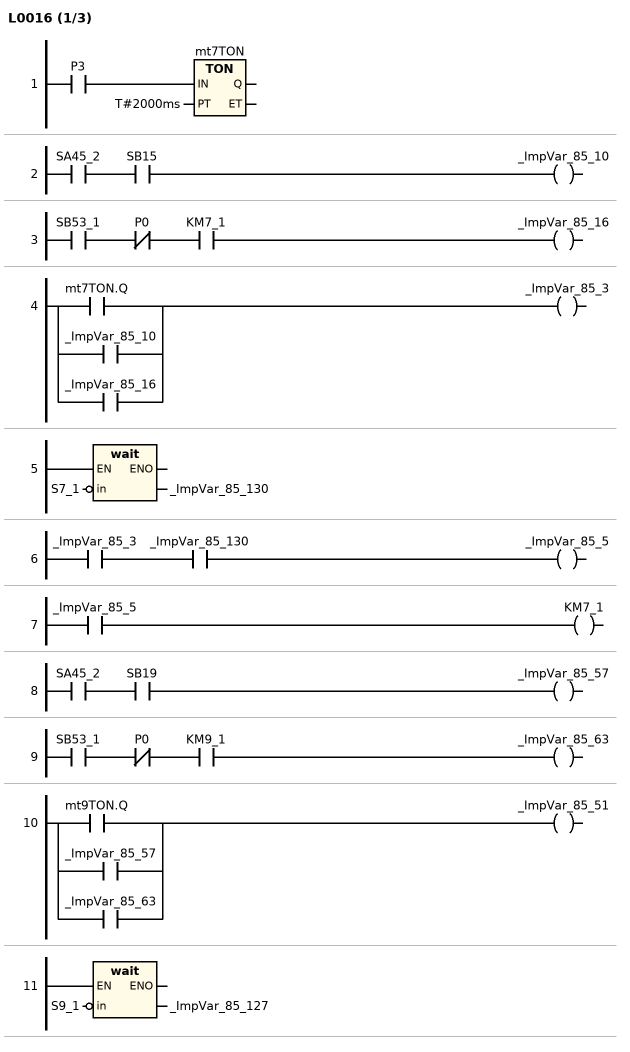
[picture p24: L0016 (LD)]
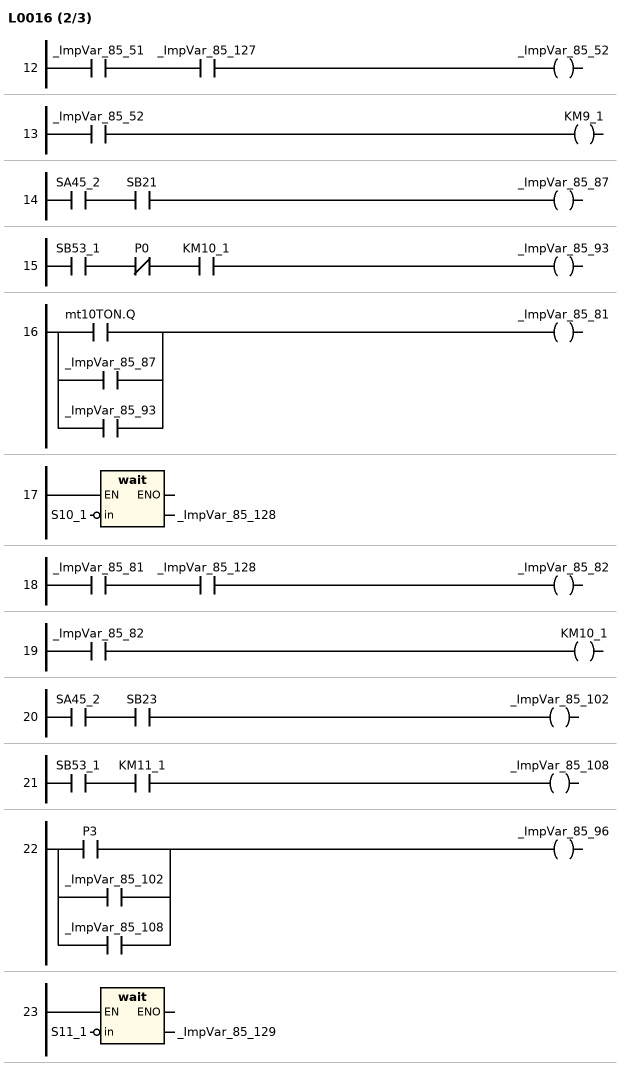
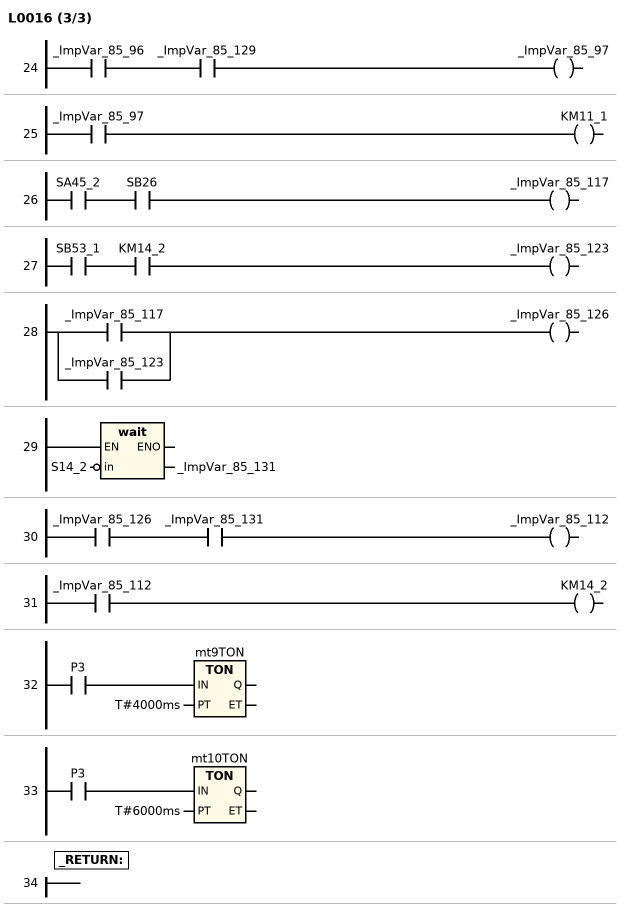
_LD_ (* Ladder Diagram *)
NETWORK 1
	[P3] - mt7TON:TON(IN: *, PT: T#2000ms)
NETWORK 2
	[SA45_2] - [SB15] --- (_ImpVar_85_10)
NETWORK 3
	[SB53_1] - [/P0] - [KM7_1] --- (_ImpVar_85_16)
NETWORK 4
	{ [mt7TON.Q] | [_ImpVar_85_10] | [_ImpVar_85_16] } --- (_ImpVar_85_3)
NETWORK 5
	*
		EN --- wait(in: NOT S7_1) => _ImpVar_85_130
NETWORK 6
	[_ImpVar_85_3] - [_ImpVar_85_130] --- (_ImpVar_85_5)
NETWORK 7
	[_ImpVar_85_5] --- (KM7_1)
NETWORK 8
	[SA45_2] - [SB19] --- (_ImpVar_85_57)
NETWORK 9
	[SB53_1] - [/P0] - [KM9_1] --- (_ImpVar_85_63)
NETWORK 10
	{ [mt9TON.Q] | [_ImpVar_85_57] | [_ImpVar_85_63] } --- (_ImpVar_85_51)
NETWORK 11
	*
		EN --- wait(in: NOT S9_1) => _ImpVar_85_127
NETWORK 12
	[_ImpVar_85_51] - [_ImpVar_85_127] --- (_ImpVar_85_52)
NETWORK 13
	[_ImpVar_85_52] --- (KM9_1)
NETWORK 14
	[SA45_2] - [SB21] --- (_ImpVar_85_87)
NETWORK 15
	[SB53_1] - [/P0] - [KM10_1] --- (_ImpVar_85_93)
NETWORK 16
	{ [mt10TON.Q] | [_ImpVar_85_87] | [_ImpVar_85_93] } --- (_ImpVar_85_81)
NETWORK 17
	*
		EN --- wait(in: NOT S10_1) => _ImpVar_85_128
NETWORK 18
	[_ImpVar_85_81] - [_ImpVar_85_128] --- (_ImpVar_85_82)
NETWORK 19
	[_ImpVar_85_82] --- (KM10_1)
NETWORK 20
	[SA45_2] - [SB23] --- (_ImpVar_85_102)
NETWORK 21
	[SB53_1] - [KM11_1] --- (_ImpVar_85_108)
NETWORK 22
	{ [P3] | [_ImpVar_85_102] | [_ImpVar_85_108] } --- (_ImpVar_85_96)
NETWORK 23
	*
		EN --- wait(in: NOT S11_1) => _ImpVar_85_129
NETWORK 24
	[_ImpVar_85_96] - [_ImpVar_85_129] --- (_ImpVar_85_97)
NETWORK 25
	[_ImpVar_85_97] --- (KM11_1)
NETWORK 26
	[SA45_2] - [SB26] --- (_ImpVar_85_117)
NETWORK 27
	[SB53_1] - [KM14_2] --- (_ImpVar_85_123)
NETWORK 28
	{ [_ImpVar_85_117] | [_ImpVar_85_123] } --- (_ImpVar_85_126)
NETWORK 29
	*
		EN --- wait(in: NOT S14_2) => _ImpVar_85_131
NETWORK 30
	[_ImpVar_85_126] - [_ImpVar_85_131] --- (_ImpVar_85_112)
NETWORK 31
	[_ImpVar_85_112] --- (KM14_2)
NETWORK 32
	[P3] - mt9TON:TON(IN: *, PT: T#4000ms)
NETWORK 33
	[P3] - mt10TON:TON(IN: *, PT: T#6000ms)
NETWORK 34 _RETURN::
	*
_END_LD_
(* the same logic as Structured Text *)
(* Network 1 *)
mt7TON(IN := P3, PT := T#2000ms);
(* Network 2 *)
_ImpVar_85_10 := SA45_2 AND SB15;
(* Network 3 *)
_ImpVar_85_16 := SB53_1 AND NOT P0 AND KM7_1;
(* Network 4 *)
_ImpVar_85_3 := mt7TON.Q OR _ImpVar_85_10 OR _ImpVar_85_16;
(* Network 5 *)
_ImpVar_85_130 := wait(in := NOT S7_1);
(* Network 6 *)
_ImpVar_85_5 := _ImpVar_85_3 AND _ImpVar_85_130;
(* Network 7 *)
KM7_1 := _ImpVar_85_5;
(* Network 8 *)
_ImpVar_85_57 := SA45_2 AND SB19;
(* Network 9 *)
_ImpVar_85_63 := SB53_1 AND NOT P0 AND KM9_1;
(* Network 10 *)
_ImpVar_85_51 := mt9TON.Q OR _ImpVar_85_57 OR _ImpVar_85_63;
(* Network 11 *)
_ImpVar_85_127 := wait(in := NOT S9_1);
(* Network 12 *)
_ImpVar_85_52 := _ImpVar_85_51 AND _ImpVar_85_127;
(* Network 13 *)
KM9_1 := _ImpVar_85_52;
(* Network 14 *)
_ImpVar_85_87 := SA45_2 AND SB21;
(* Network 15 *)
_ImpVar_85_93 := SB53_1 AND NOT P0 AND KM10_1;
(* Network 16 *)
_ImpVar_85_81 := mt10TON.Q OR _ImpVar_85_87 OR _ImpVar_85_93;
(* Network 17 *)
_ImpVar_85_128 := wait(in := NOT S10_1);
(* Network 18 *)
_ImpVar_85_82 := _ImpVar_85_81 AND _ImpVar_85_128;
(* Network 19 *)
KM10_1 := _ImpVar_85_82;
(* Network 20 *)
_ImpVar_85_102 := SA45_2 AND SB23;
(* Network 21 *)
_ImpVar_85_108 := SB53_1 AND KM11_1;
(* Network 22 *)
_ImpVar_85_96 := P3 OR _ImpVar_85_102 OR _ImpVar_85_108;
(* Network 23 *)
_ImpVar_85_129 := wait(in := NOT S11_1);
(* Network 24 *)
_ImpVar_85_97 := _ImpVar_85_96 AND _ImpVar_85_129;
(* Network 25 *)
KM11_1 := _ImpVar_85_97;
(* Network 26 *)
_ImpVar_85_117 := SA45_2 AND SB26;
(* Network 27 *)
_ImpVar_85_123 := SB53_1 AND KM14_2;
(* Network 28 *)
_ImpVar_85_126 := _ImpVar_85_117 OR _ImpVar_85_123;
(* Network 29 *)
_ImpVar_85_131 := wait(in := NOT S14_2);
(* Network 30 *)
_ImpVar_85_112 := _ImpVar_85_126 AND _ImpVar_85_131;
(* Network 31 *)
KM14_2 := _ImpVar_85_112;
(* Network 32 *)
mt9TON(IN := P3, PT := T#4000ms);
(* Network 33 *)
mt10TON(IN := P3, PT := T#6000ms);
(* Network 34 *)
(* label: _RETURN: *)
END_PROGRAM

(* POU gatesAlarm, LD *)
PROGRAM gatesAlarm
VAR
	al1: alarm;
	al18_2: alarm;
	al18_1: alarm;
	al4_1: alarm;
	al4_2: alarm;
	al5_1: alarm;
	al5_2: alarm;
	al6_1: alarm;
	al6_2: alarm;
	al7_2: alarm;
	al7_1: alarm;
	al8_1: alarm;
	al8_2: alarm;
	al9_1: alarm;
	al9_2: alarm;
	al10_1: alarm;
	al10_2: alarm;
	a11_1: alarm;
	al11_2: alarm;
	al14_1: alarm;
	al14_2: alarm;
	vaqt : WORD := 70;
END_VAR
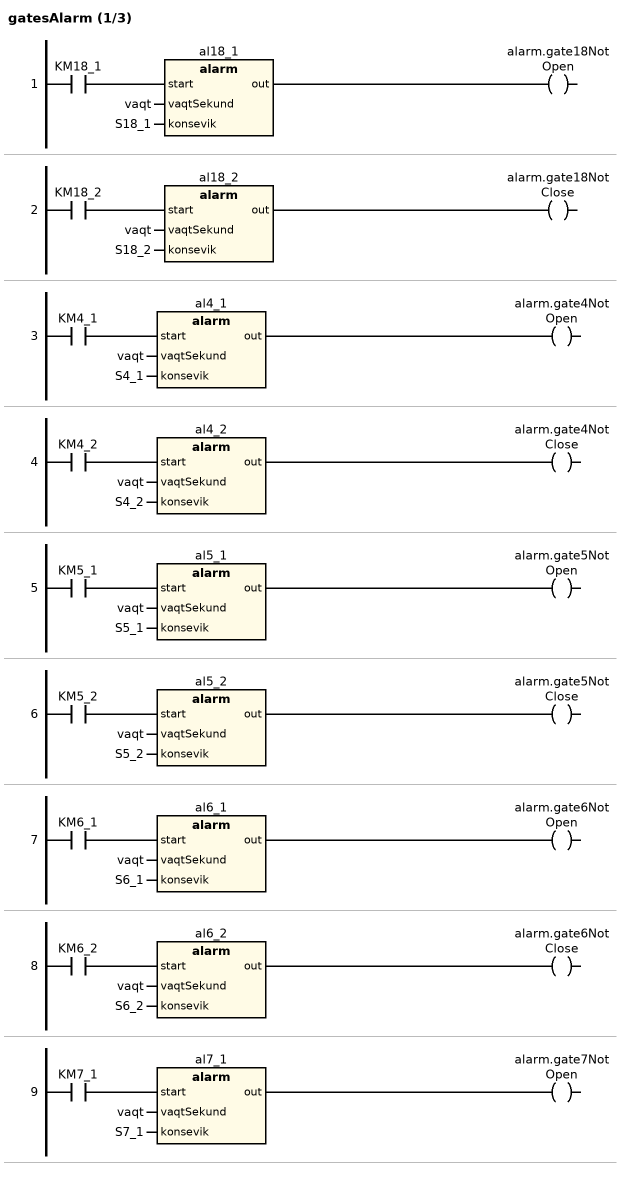
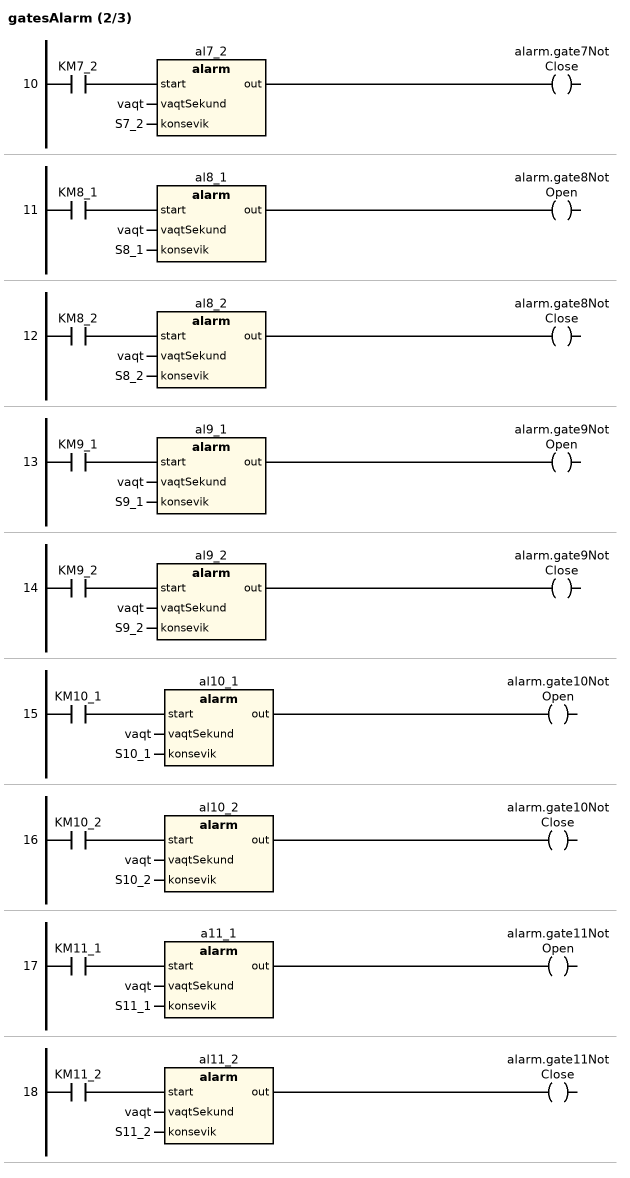
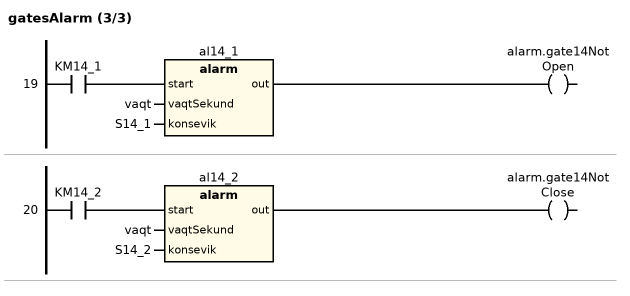
_LD_ (* Ladder Diagram *)
NETWORK 1
	[KM18_1] - al18_1:alarm(start: *, vaqtSekund: vaqt, konsevik: S18_1) --- (alarm.gate18NotOpen)
NETWORK 2
	[KM18_2] - al18_2:alarm(start: *, vaqtSekund: vaqt, konsevik: S18_2) --- (alarm.gate18NotClose)
NETWORK 3
	[KM4_1] - al4_1:alarm(start: *, vaqtSekund: vaqt, konsevik: S4_1) --- (alarm.gate4NotOpen)
NETWORK 4
	[KM4_2] - al4_2:alarm(start: *, vaqtSekund: vaqt, konsevik: S4_2) --- (alarm.gate4NotClose)
NETWORK 5
	[KM5_1] - al5_1:alarm(start: *, vaqtSekund: vaqt, konsevik: S5_1) --- (alarm.gate5NotOpen)
NETWORK 6
	[KM5_2] - al5_2:alarm(start: *, vaqtSekund: vaqt, konsevik: S5_2) --- (alarm.gate5NotClose)
NETWORK 7
	[KM6_1] - al6_1:alarm(start: *, vaqtSekund: vaqt, konsevik: S6_1) --- (alarm.gate6NotOpen)
NETWORK 8
	[KM6_2] - al6_2:alarm(start: *, vaqtSekund: vaqt, konsevik: S6_2) --- (alarm.gate6NotClose)
NETWORK 9
	[KM7_1] - al7_1:alarm(start: *, vaqtSekund: vaqt, konsevik: S7_1) --- (alarm.gate7NotOpen)
NETWORK 10
	[KM7_2] - al7_2:alarm(start: *, vaqtSekund: vaqt, konsevik: S7_2) --- (alarm.gate7NotClose)
NETWORK 11
	[KM8_1] - al8_1:alarm(start: *, vaqtSekund: vaqt, konsevik: S8_1) --- (alarm.gate8NotOpen)
NETWORK 12
	[KM8_2] - al8_2:alarm(start: *, vaqtSekund: vaqt, konsevik: S8_2) --- (alarm.gate8NotClose)
NETWORK 13
	[KM9_1] - al9_1:alarm(start: *, vaqtSekund: vaqt, konsevik: S9_1) --- (alarm.gate9NotOpen)
NETWORK 14
	[KM9_2] - al9_2:alarm(start: *, vaqtSekund: vaqt, konsevik: S9_2) --- (alarm.gate9NotClose)
NETWORK 15
	[KM10_1] - al10_1:alarm(start: *, vaqtSekund: vaqt, konsevik: S10_1) --- (alarm.gate10NotOpen)
NETWORK 16
	[KM10_2] - al10_2:alarm(start: *, vaqtSekund: vaqt, konsevik: S10_2) --- (alarm.gate10NotClose)
NETWORK 17
	[KM11_1] - a11_1:alarm(start: *, vaqtSekund: vaqt, konsevik: S11_1) --- (alarm.gate11NotOpen)
NETWORK 18
	[KM11_2] - al11_2:alarm(start: *, vaqtSekund: vaqt, konsevik: S11_2) --- (alarm.gate11NotClose)
NETWORK 19
	[KM14_1] - al14_1:alarm(start: *, vaqtSekund: vaqt, konsevik: S14_1) --- (alarm.gate14NotOpen)
NETWORK 20
	[KM14_2] - al14_2:alarm(start: *, vaqtSekund: vaqt, konsevik: S14_2) --- (alarm.gate14NotClose)
_END_LD_
(* the same logic as Structured Text *)
(* Network 1 *)
al18_1(start := KM18_1, vaqtSekund := vaqt, konsevik := S18_1);
alarm.gate18NotOpen := al18_1.out;
(* Network 2 *)
al18_2(start := KM18_2, vaqtSekund := vaqt, konsevik := S18_2);
alarm.gate18NotClose := al18_2.out;
(* Network 3 *)
al4_1(start := KM4_1, vaqtSekund := vaqt, konsevik := S4_1);
alarm.gate4NotOpen := al4_1.out;
(* Network 4 *)
al4_2(start := KM4_2, vaqtSekund := vaqt, konsevik := S4_2);
alarm.gate4NotClose := al4_2.out;
(* Network 5 *)
al5_1(start := KM5_1, vaqtSekund := vaqt, konsevik := S5_1);
alarm.gate5NotOpen := al5_1.out;
(* Network 6 *)
al5_2(start := KM5_2, vaqtSekund := vaqt, konsevik := S5_2);
alarm.gate5NotClose := al5_2.out;
(* Network 7 *)
al6_1(start := KM6_1, vaqtSekund := vaqt, konsevik := S6_1);
alarm.gate6NotOpen := al6_1.out;
(* Network 8 *)
al6_2(start := KM6_2, vaqtSekund := vaqt, konsevik := S6_2);
alarm.gate6NotClose := al6_2.out;
(* Network 9 *)
al7_1(start := KM7_1, vaqtSekund := vaqt, konsevik := S7_1);
alarm.gate7NotOpen := al7_1.out;
(* Network 10 *)
al7_2(start := KM7_2, vaqtSekund := vaqt, konsevik := S7_2);
alarm.gate7NotClose := al7_2.out;
(* Network 11 *)
al8_1(start := KM8_1, vaqtSekund := vaqt, konsevik := S8_1);
alarm.gate8NotOpen := al8_1.out;
(* Network 12 *)
al8_2(start := KM8_2, vaqtSekund := vaqt, konsevik := S8_2);
alarm.gate8NotClose := al8_2.out;
(* Network 13 *)
al9_1(start := KM9_1, vaqtSekund := vaqt, konsevik := S9_1);
alarm.gate9NotOpen := al9_1.out;
(* Network 14 *)
al9_2(start := KM9_2, vaqtSekund := vaqt, konsevik := S9_2);
alarm.gate9NotClose := al9_2.out;
(* Network 15 *)
al10_1(start := KM10_1, vaqtSekund := vaqt, konsevik := S10_1);
alarm.gate10NotOpen := al10_1.out;
(* Network 16 *)
al10_2(start := KM10_2, vaqtSekund := vaqt, konsevik := S10_2);
alarm.gate10NotClose := al10_2.out;
(* Network 17 *)
a11_1(start := KM11_1, vaqtSekund := vaqt, konsevik := S11_1);
alarm.gate11NotOpen := a11_1.out;
(* Network 18 *)
al11_2(start := KM11_2, vaqtSekund := vaqt, konsevik := S11_2);
alarm.gate11NotClose := al11_2.out;
(* Network 19 *)
al14_1(start := KM14_1, vaqtSekund := vaqt, konsevik := S14_1);
alarm.gate14NotOpen := al14_1.out;
(* Network 20 *)
al14_2(start := KM14_2, vaqtSekund := vaqt, konsevik := S14_2);
alarm.gate14NotClose := al14_2.out;
END_PROGRAM

(* POU start_or_stop, LD *)
PROGRAM start_or_stop
VAR
	_controlFazaDI46: BOOL;
	kompressorOFF: TP;
	kompressorON: TP;
	_currentHighJD5DI00000: BOOL;
	P300000: BOOL;
	P00000: BOOL;

	alarmLedDO_MB555: BOOL;
	_kompOffDO_55555555: BOOL;
	_kompOnDO_555555: BOOL;
	trig: R_TRIG;

END_VAR
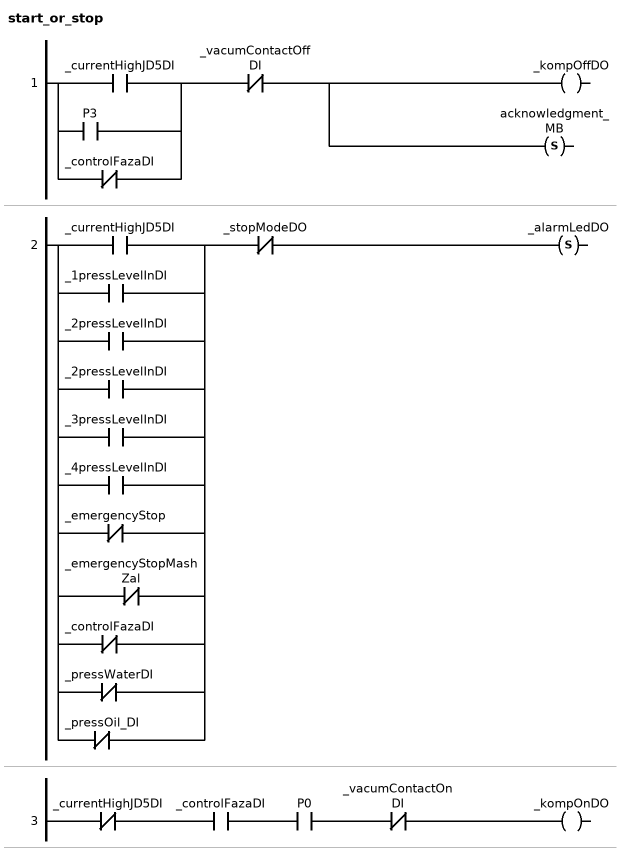
_LD_ (* Ladder Diagram *)
NETWORK 1
	{ [_currentHighJD5DI] | [P3] | [/_controlFazaDI] } - [/_vacumContactOffDI] --- (_kompOffDO) (S acknowledgment_MB)
NETWORK 2
	{ [_currentHighJD5DI] | [_1pressLevelInDI] | [_2pressLevelInDI] | [_2pressLevelInDI] | [_3pressLevelInDI] | [_4pressLevelInDI] | [/_emergencyStop] | [/_emergencyStopMashZal] | [/_controlFazaDI] | [/_pressWaterDI] | [/_pressOil_DI] } - [/_stopModeDO] --- (S _alarmLedDO)
NETWORK 3
	[/_currentHighJD5DI] - [_controlFazaDI] - [P0] - [/_vacumContactOnDI] --- (_kompOnDO)
_END_LD_
(* the same logic as Structured Text *)
(* Network 1 *)
_kompOffDO := (_currentHighJD5DI OR P3 OR NOT _controlFazaDI) AND NOT _vacumContactOffDI;
IF _kompOffDO THEN acknowledgment_MB := TRUE; END_IF;
(* Network 2 *)
IF (_currentHighJD5DI OR _1pressLevelInDI OR _2pressLevelInDI OR _2pressLevelInDI OR _3pressLevelInDI OR _4pressLevelInDI OR NOT _emergencyStop OR NOT _emergencyStopMashZal OR NOT _controlFazaDI OR NOT _pressWaterDI OR NOT _pressOil_DI) AND NOT _stopModeDO THEN _alarmLedDO := TRUE; END_IF;
(* Network 3 *)
_kompOnDO := NOT _currentHighJD5DI AND _controlFazaDI AND P0 AND NOT _vacumContactOnDI;
END_PROGRAM

(* POU E_STOP, LD *)
PROGRAM E_STOP
VAR
	P4: BOOL;
	tof1: TON;
	rtrig: R_TRIG;
	xato : ARRAY [0..17] OF BOOL;
	ton1 : TON;
END_VAR
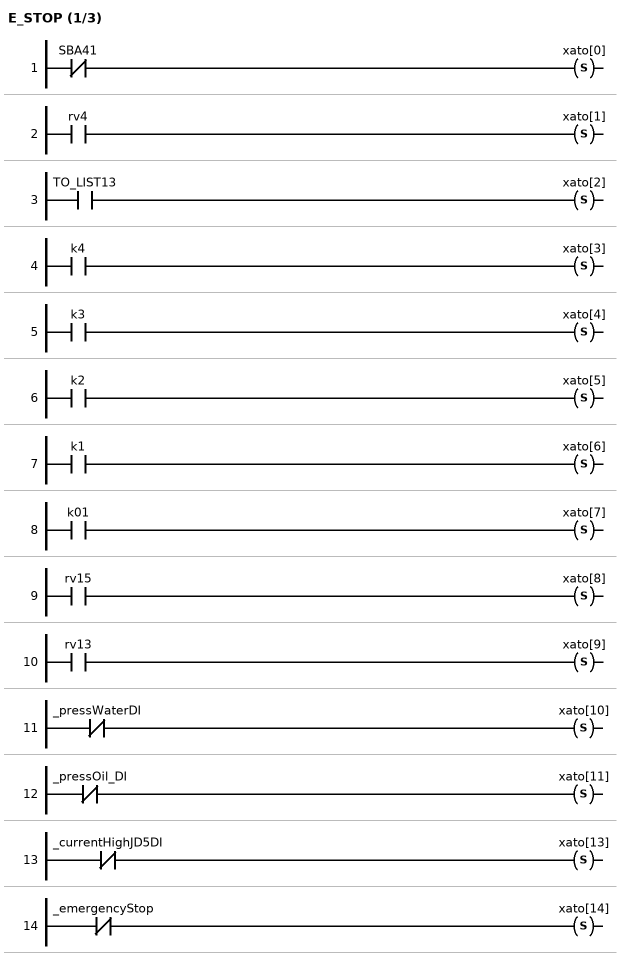
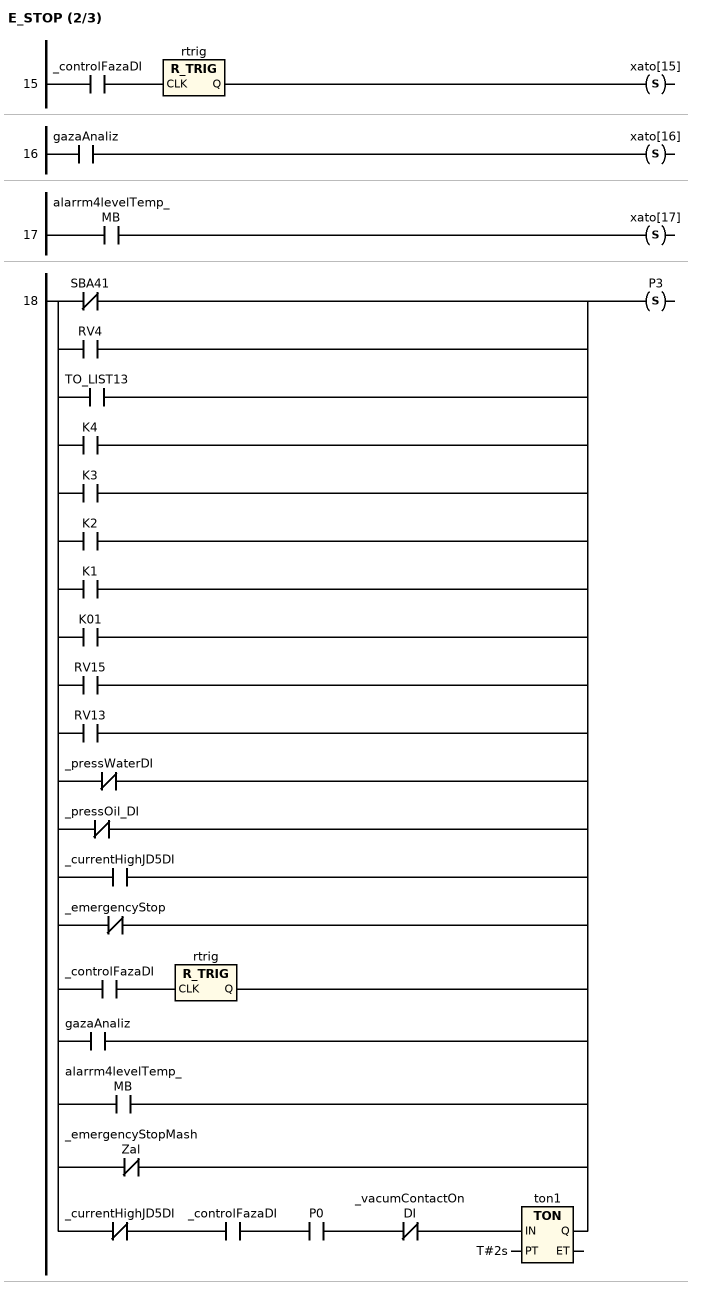
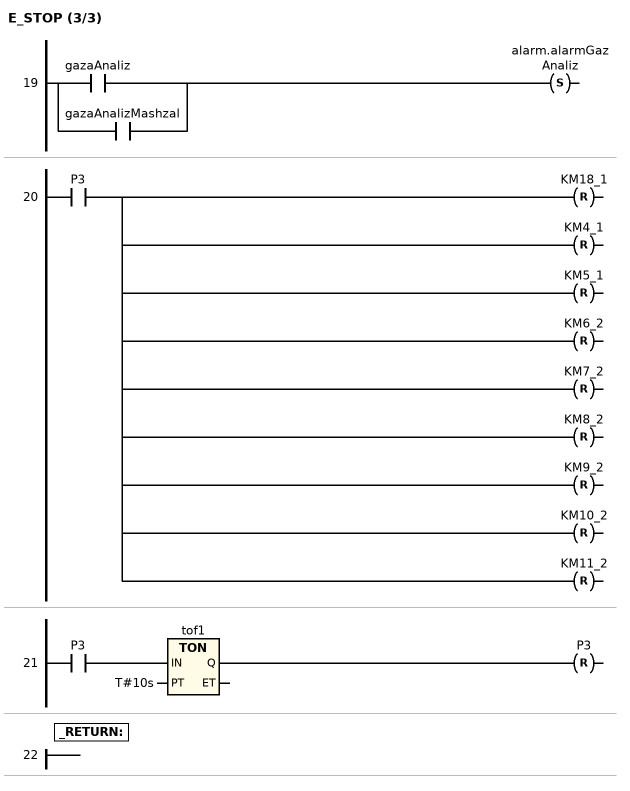
_LD_ (* Ladder Diagram *)
NETWORK 1
	[/SBA41] --- (S xato[0])
NETWORK 2
	[rv4] --- (S xato[1])
NETWORK 3
	[TO_LIST13] --- (S xato[2])
NETWORK 4
	[k4] --- (S xato[3])
NETWORK 5
	[k3] --- (S xato[4])
NETWORK 6
	[k2] --- (S xato[5])
NETWORK 7
	[k1] --- (S xato[6])
NETWORK 8
	[k01] --- (S xato[7])
NETWORK 9
	[rv15] --- (S xato[8])
NETWORK 10
	[rv13] --- (S xato[9])
NETWORK 11
	[/_pressWaterDI] --- (S xato[10])
NETWORK 12
	[/_pressOil_DI] --- (S xato[11])
NETWORK 13
	[/_currentHighJD5DI] --- (S xato[13])
NETWORK 14
	[/_emergencyStop] --- (S xato[14])
NETWORK 15
	[_controlFazaDI] - rtrig:R_TRIG(CLK: *) --- (S xato[15])
NETWORK 16
	[gazaAnaliz] --- (S xato[16])
NETWORK 17
	[alarrm4levelTemp_MB] --- (S xato[17])
NETWORK 18
	{ [/SBA41] | [RV4] | [TO_LIST13] | [K4] | [K3] | [K2] | [K1] | [K01] | [RV15] | [RV13] | [/_pressWaterDI] | [/_pressOil_DI] | [_currentHighJD5DI] | [/_emergencyStop] | [_controlFazaDI] - rtrig:R_TRIG(CLK: *) | [gazaAnaliz] | [alarrm4levelTemp_MB] | [/_emergencyStopMashZal] | [/_currentHighJD5DI] - [_controlFazaDI] - [P0] - [/_vacumContactOnDI] - ton1:TON(IN: *, PT: T#2s) } --- (S P3)
NETWORK 19
	{ [gazaAnaliz] | [gazaAnalizMashzal] } --- (S alarm.alarmGazAnaliz)
NETWORK 20
	[P3] --- (R KM18_1) (R KM4_1) (R KM5_1) (R KM6_2) (R KM7_2) (R KM8_2) (R KM9_2) (R KM10_2) (R KM11_2)
NETWORK 21
	[P3] - tof1:TON(IN: *, PT: T#10s) --- (R P3)
NETWORK 22 _RETURN::
	*
_END_LD_
(* the same logic as Structured Text *)
(* Network 1 *)
IF NOT SBA41 THEN xato[0] := TRUE; END_IF;
(* Network 2 *)
IF rv4 THEN xato[1] := TRUE; END_IF;
(* Network 3 *)
IF TO_LIST13 THEN xato[2] := TRUE; END_IF;
(* Network 4 *)
IF k4 THEN xato[3] := TRUE; END_IF;
(* Network 5 *)
IF k3 THEN xato[4] := TRUE; END_IF;
(* Network 6 *)
IF k2 THEN xato[5] := TRUE; END_IF;
(* Network 7 *)
IF k1 THEN xato[6] := TRUE; END_IF;
(* Network 8 *)
IF k01 THEN xato[7] := TRUE; END_IF;
(* Network 9 *)
IF rv15 THEN xato[8] := TRUE; END_IF;
(* Network 10 *)
IF rv13 THEN xato[9] := TRUE; END_IF;
(* Network 11 *)
IF NOT _pressWaterDI THEN xato[10] := TRUE; END_IF;
(* Network 12 *)
IF NOT _pressOil_DI THEN xato[11] := TRUE; END_IF;
(* Network 13 *)
IF NOT _currentHighJD5DI THEN xato[13] := TRUE; END_IF;
(* Network 14 *)
IF NOT _emergencyStop THEN xato[14] := TRUE; END_IF;
(* Network 15 *)
rtrig(CLK := _controlFazaDI);
IF rtrig.Q THEN xato[15] := TRUE; END_IF;
(* Network 16 *)
IF gazaAnaliz THEN xato[16] := TRUE; END_IF;
(* Network 17 *)
IF alarrm4levelTemp_MB THEN xato[17] := TRUE; END_IF;
(* Network 18 *)
rtrig(CLK := _controlFazaDI);
ton1(IN := NOT _currentHighJD5DI AND _controlFazaDI AND P0 AND NOT _vacumContactOnDI, PT := T#2s);
IF NOT SBA41 OR RV4 OR TO_LIST13 OR K4 OR K3 OR K2 OR K1 OR K01 OR RV15 OR RV13 OR NOT _pressWaterDI OR NOT _pressOil_DI OR _currentHighJD5DI OR NOT _emergencyStop OR rtrig.Q OR gazaAnaliz OR alarrm4levelTemp_MB OR NOT _emergencyStopMashZal OR ton1.Q THEN P3 := TRUE; END_IF;
(* Network 19 *)
IF gazaAnaliz OR gazaAnalizMashzal THEN alarm.alarmGazAnaliz := TRUE; END_IF;
(* Network 20 *)
IF P3 THEN KM18_1 := FALSE; KM4_1 := FALSE; KM5_1 := FALSE; KM6_2 := FALSE; KM7_2 := FALSE; KM8_2 := FALSE; KM9_2 := FALSE; KM10_2 := FALSE; KM11_2 := FALSE; END_IF;
(* Network 21 *)
tof1(IN := P3, PT := T#10s);
IF tof1.Q THEN P3 := FALSE; END_IF;
(* Network 22 *)
(* label: _RETURN: *)
END_PROGRAM

(* POU blink, CFC *)
PROGRAM blink
VAR
	tp1: TP;
	tp2: TP;
	out: BOOL;
	vaqt : TIME := T#500ms;
END_VAR
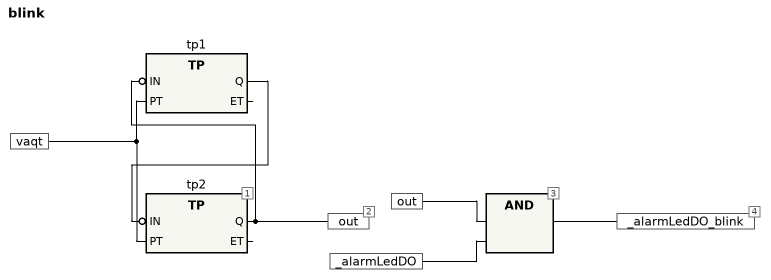
_CFC_ (* Continuous Function Chart, elements in execution order *)
#0 tp1:TP(IN: NOT #1.Q, PT: vaqt)
#1 tp2:TP(IN: NOT #0.Q, PT: vaqt)
#2 out <= #1.Q
#3 AND(out, _alarmLedDO)
#4 _alarmLedDO_blink <= #3
_END_CFC_
(* the same logic as Structured Text *)
tp1(IN := NOT tp2.Q, PT := vaqt);
tp2(IN := NOT tp1.Q, PT := vaqt);
out := tp2.Q;
_alarmLedDO_blink := out AND _alarmLedDO;
END_PROGRAM

(* POU L005, CFC *)
PROGRAM L005
VAR
	_kompOffDO000000000: BOOL;
	t6AfterTON : TON;

END_VAR
VAR (* helpers for the ST form of the networks *)
	_t5 : BOOL;
	_t6 : BOOL;
	_t36 : BOOL;
	_t141 : BOOL;
	_t46 : BOOL;
END_VAR
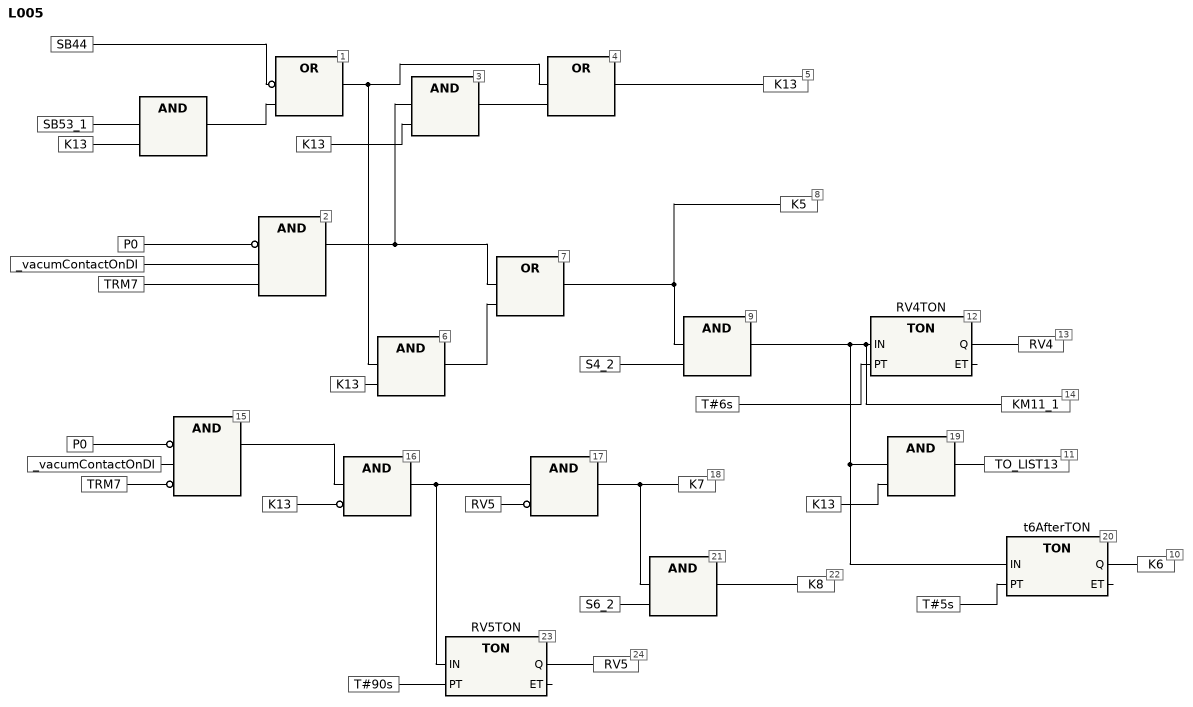
_CFC_ (* Continuous Function Chart, elements in execution order *)
#0 AND(SB53_1, K13)
#1 OR(NOT SB44, #0)
#2 AND(NOT P0, _vacumContactOnDI, TRM7)
#3 AND(#2, K13)
#4 OR(#1, #3)
#5 K13 <= #4
#6 AND(#1, K13)
#7 OR(#2, #6)
#8 K5 <= #7
#9 AND(#7, S4_2)
#10 K6 <= #20.Q
#11 TO_LIST13 <= #19
#12 RV4TON:TON(IN: #9, PT: T#6s)
#13 RV4 <= #12.Q
#14 KM11_1 <= #9
#15 AND(NOT P0, _vacumContactOnDI, NOT TRM7)
#16 AND(#15, NOT K13)
#17 AND(#16, NOT RV5)
#18 K7 <= #17
#19 AND(#9, K13)
#20 t6AfterTON:TON(IN: #9, PT: T#5s)
#21 AND(#17, S6_2)
#22 K8 <= #21
#23 RV5TON:TON(IN: #16, PT: T#90s)
#24 RV5 <= #23.Q
_END_CFC_
(* the same logic as Structured Text *)
_t5 := NOT SB44 OR (SB53_1 AND K13);
_t6 := NOT P0 AND _vacumContactOnDI AND TRM7;
K13 := _t5 OR (_t6 AND K13);
K5 := _t6 OR (_t5 AND K13);
_t36 := (_t6 OR (_t5 AND K13)) AND S4_2;
K6 := t6AfterTON.Q;
TO_LIST13 := _t141;
RV4TON(IN := _t36, PT := T#6s);
RV4 := RV4TON.Q;
KM11_1 := _t36;
_t46 := (NOT P0 AND _vacumContactOnDI AND NOT TRM7) AND NOT K13;
K7 := _t46 AND NOT RV5;
_t141 := _t36 AND K13;
t6AfterTON(IN := _t36, PT := T#5s);
K8 := (_t46 AND NOT RV5) AND S6_2;
RV5TON(IN := _t46, PT := T#90s);
RV5 := RV5TON.Q;
END_PROGRAM

(* POU L008, CFC *)
PROGRAM L008
VAR


END_VAR
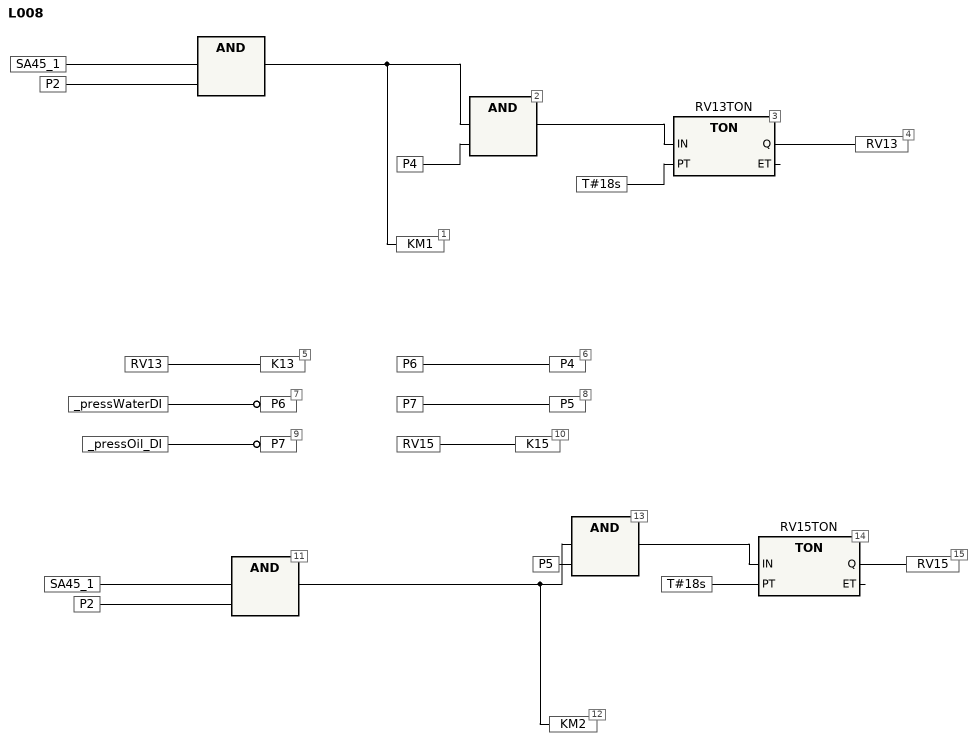
_CFC_ (* Continuous Function Chart, elements in execution order *)
#0 AND(SA45_1, P2)
#1 KM1 <= #0
#2 AND(#0, P4)
#3 RV13TON:TON(IN: #2, PT: T#18s)
#4 RV13 <= #3.Q
#5 K13 <= RV13
#6 P4 <= P6
#7 P6 <= NOT _pressWaterDI
#8 P5 <= P7
#9 P7 <= NOT _pressOil_DI
#10 K15 <= RV15
#11 AND(SA45_1, P2)
#12 KM2 <= #11
#13 AND(#11, P5)
#14 RV15TON:TON(IN: #13, PT: T#18s)
#15 RV15 <= #14.Q
_END_CFC_
(* the same logic as Structured Text *)
KM1 := SA45_1 AND P2;
RV13TON(IN := (SA45_1 AND P2) AND P4, PT := T#18s);
RV13 := RV13TON.Q;
K13 := RV13;
P4 := P6;
P6 := NOT _pressWaterDI;
P5 := P7;
P7 := NOT _pressOil_DI;
K15 := RV15;
KM2 := SA45_1 AND P2;
RV15TON(IN := (SA45_1 AND P2) AND P5, PT := T#18s);
RV15 := RV15TON.Q;
END_PROGRAM

(* POU L009, CFC *)
PROGRAM L009
VAR




	S18_1_prymoy: BOOL := TRUE;
END_VAR
VAR (* helpers for the ST form of the networks *)
	_t49 : BOOL;
END_VAR
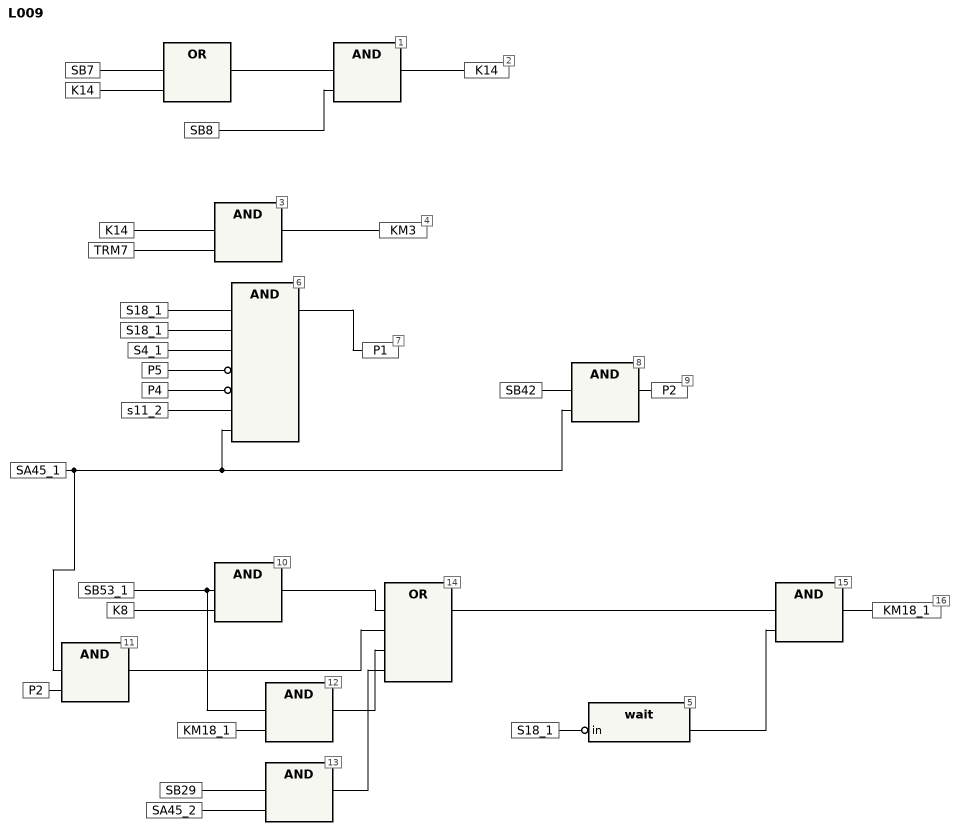
_CFC_ (* Continuous Function Chart, elements in execution order *)
#0 OR(SB7, K14)
#1 AND(#0, SB8)
#2 K14 <= #1
#3 AND(K14, TRM7)
#4 KM3 <= #3
#5 wait(in: NOT S18_1)
#6 AND(S18_1, S18_1, S4_1, NOT P5, NOT P4, s11_2, SA45_1)
#7 P1 <= #6
#8 AND(SB42, SA45_1)
#9 P2 <= #8
#10 AND(SB53_1, K8)
#11 AND(SA45_1, P2)
#12 AND(SB53_1, KM18_1)
#13 AND(SB29, SA45_2)
#14 OR(#10, #11, #12, #13)
#15 AND(#14, #5)
#16 KM18_1 <= #15
_END_CFC_
(* the same logic as Structured Text *)
K14 := (SB7 OR K14) AND SB8;
KM3 := K14 AND TRM7;
_t49 := wait(in := NOT S18_1);
P1 := S18_1 AND S18_1 AND S4_1 AND NOT P5 AND NOT P4 AND s11_2 AND SA45_1;
P2 := SB42 AND SA45_1;
KM18_1 := ((SB53_1 AND K8) OR (SA45_1 AND P2) OR (SB53_1 AND KM18_1) OR (SB29 AND SA45_2)) AND _t49;
END_PROGRAM

(* POU L010, CFC *)
PROGRAM L010
VAR
	_17S_2: BOOL;

END_VAR
VAR (* helpers for the ST form of the networks *)
	_t68 : BOOL;
	_t69 : BOOL;
END_VAR
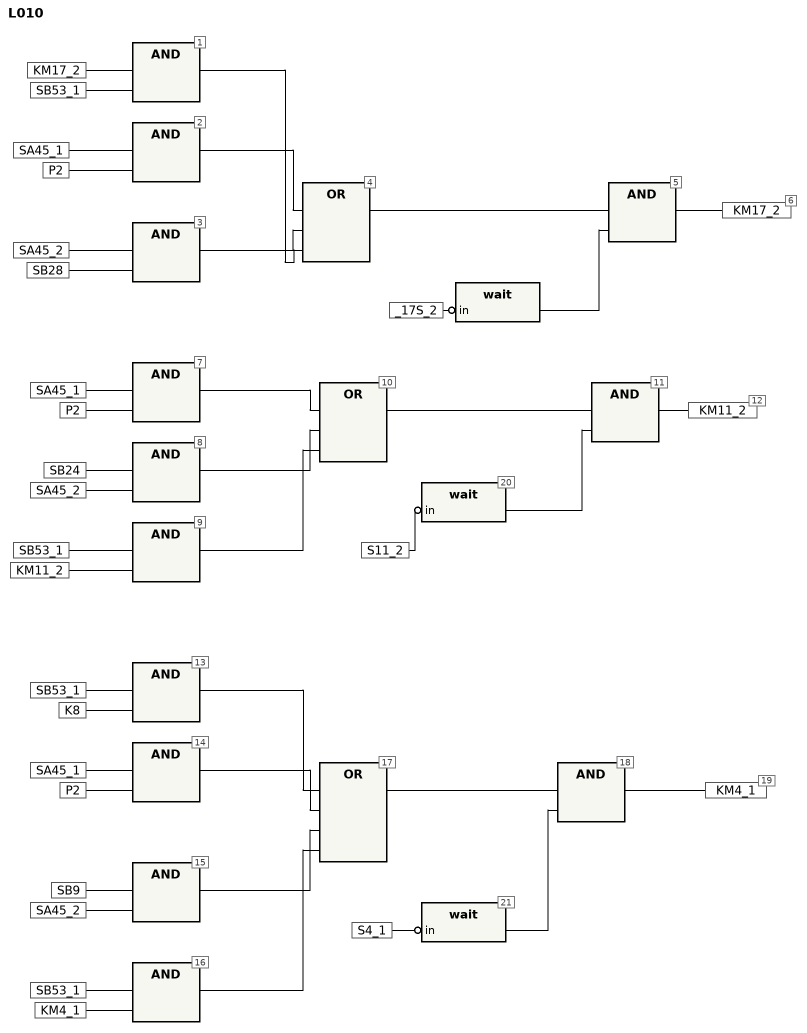
_CFC_ (* Continuous Function Chart, elements in execution order *)
#0 wait(in: NOT _17S_2)
#1 AND(KM17_2, SB53_1)
#2 AND(SA45_1, P2)
#3 AND(SA45_2, SB28)
#4 OR(#2, #3, #1)
#5 AND(#4, #0)
#6 KM17_2 <= #5
#7 AND(SA45_1, P2)
#8 AND(SB24, SA45_2)
#9 AND(SB53_1, KM11_2)
#10 OR(#7, #8, #9)
#11 AND(#10, #20)
#12 KM11_2 <= #11
#13 AND(SB53_1, K8)
#14 AND(SA45_1, P2)
#15 AND(SB9, SA45_2)
#16 AND(SB53_1, KM4_1)
#17 OR(#13, #14, #15, #16)
#18 AND(#17, #21)
#19 KM4_1 <= #18
#20 wait(in: NOT S11_2)
#21 wait(in: NOT S4_1)
_END_CFC_
(* the same logic as Structured Text *)
KM17_2 := ((SA45_1 AND P2) OR (SA45_2 AND SB28) OR (KM17_2 AND SB53_1)) AND wait(in := NOT _17S_2);
KM11_2 := ((SA45_1 AND P2) OR (SB24 AND SA45_2) OR (SB53_1 AND KM11_2)) AND _t68;
KM4_1 := ((SB53_1 AND K8) OR (SA45_1 AND P2) OR (SB9 AND SA45_2) OR (SB53_1 AND KM4_1)) AND _t69;
_t68 := wait(in := NOT S11_2);
_t69 := wait(in := NOT S4_1);
END_PROGRAM

(* POU L011, CFC *)
PROGRAM L011
VAR


	_16S_2: BOOL;
END_VAR
VAR (* helpers for the ST form of the networks *)
	_t55 : BOOL;
	_t54 : BOOL;
	_t36 : BOOL;
END_VAR
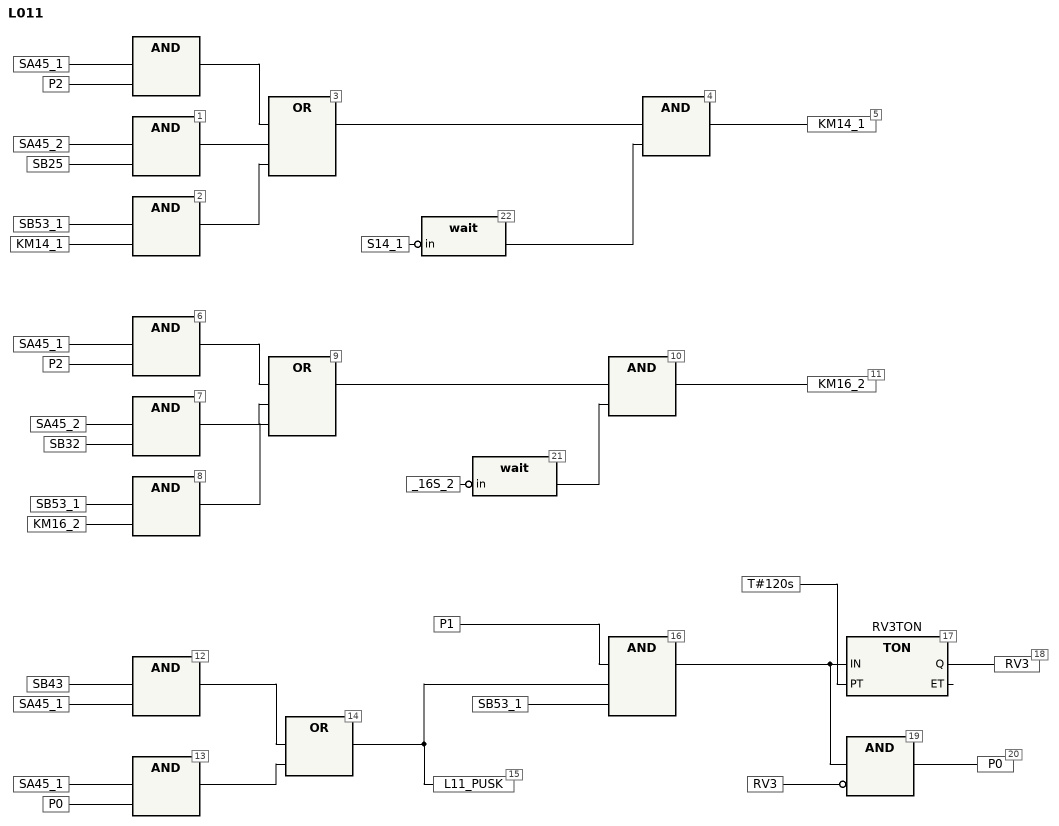
_CFC_ (* Continuous Function Chart, elements in execution order *)
#0 AND(SA45_1, P2)
#1 AND(SA45_2, SB25)
#2 AND(SB53_1, KM14_1)
#3 OR(#0, #1, #2)
#4 AND(#3, #22)
#5 KM14_1 <= #4
#6 AND(SA45_1, P2)
#7 AND(SA45_2, SB32)
#8 AND(SB53_1, KM16_2)
#9 OR(#6, #7, #8)
#10 AND(#9, #21)
#11 KM16_2 <= #10
#12 AND(SB43, SA45_1)
#13 AND(SA45_1, P0)
#14 OR(#12, #13)
#15 L11_PUSK <= #14
#16 AND(P1, #14, SB53_1)
#17 RV3TON:TON(IN: #16, PT: T#120s)
#18 RV3 <= #17.Q
#19 AND(#16, NOT RV3)
#20 P0 <= #19
#21 wait(in: NOT _16S_2)
#22 wait(in: NOT S14_1)
_END_CFC_
(* the same logic as Structured Text *)
KM14_1 := ((SA45_1 AND P2) OR (SA45_2 AND SB25) OR (SB53_1 AND KM14_1)) AND _t55;
KM16_2 := ((SA45_1 AND P2) OR (SA45_2 AND SB32) OR (SB53_1 AND KM16_2)) AND _t54;
_t36 := (SB43 AND SA45_1) OR (SA45_1 AND P0);
L11_PUSK := _t36;
RV3TON(IN := P1 AND _t36 AND SB53_1, PT := T#120s);
RV3 := RV3TON.Q;
P0 := (P1 AND _t36 AND SB53_1) AND NOT RV3;
_t54 := wait(in := NOT _16S_2);
_t55 := wait(in := NOT S14_1);
END_PROGRAM

(* POU L012, CFC *)
PROGRAM L012
VAR







END_VAR
VAR (* helpers for the ST form of the networks *)
	_t5 : BOOL;
	_t85 : BOOL;
	_t25 : BOOL;
	_t86 : BOOL;
	_t45 : BOOL;
	_t87 : BOOL;
	_t59 : BOOL;
	_t88 : BOOL;
END_VAR
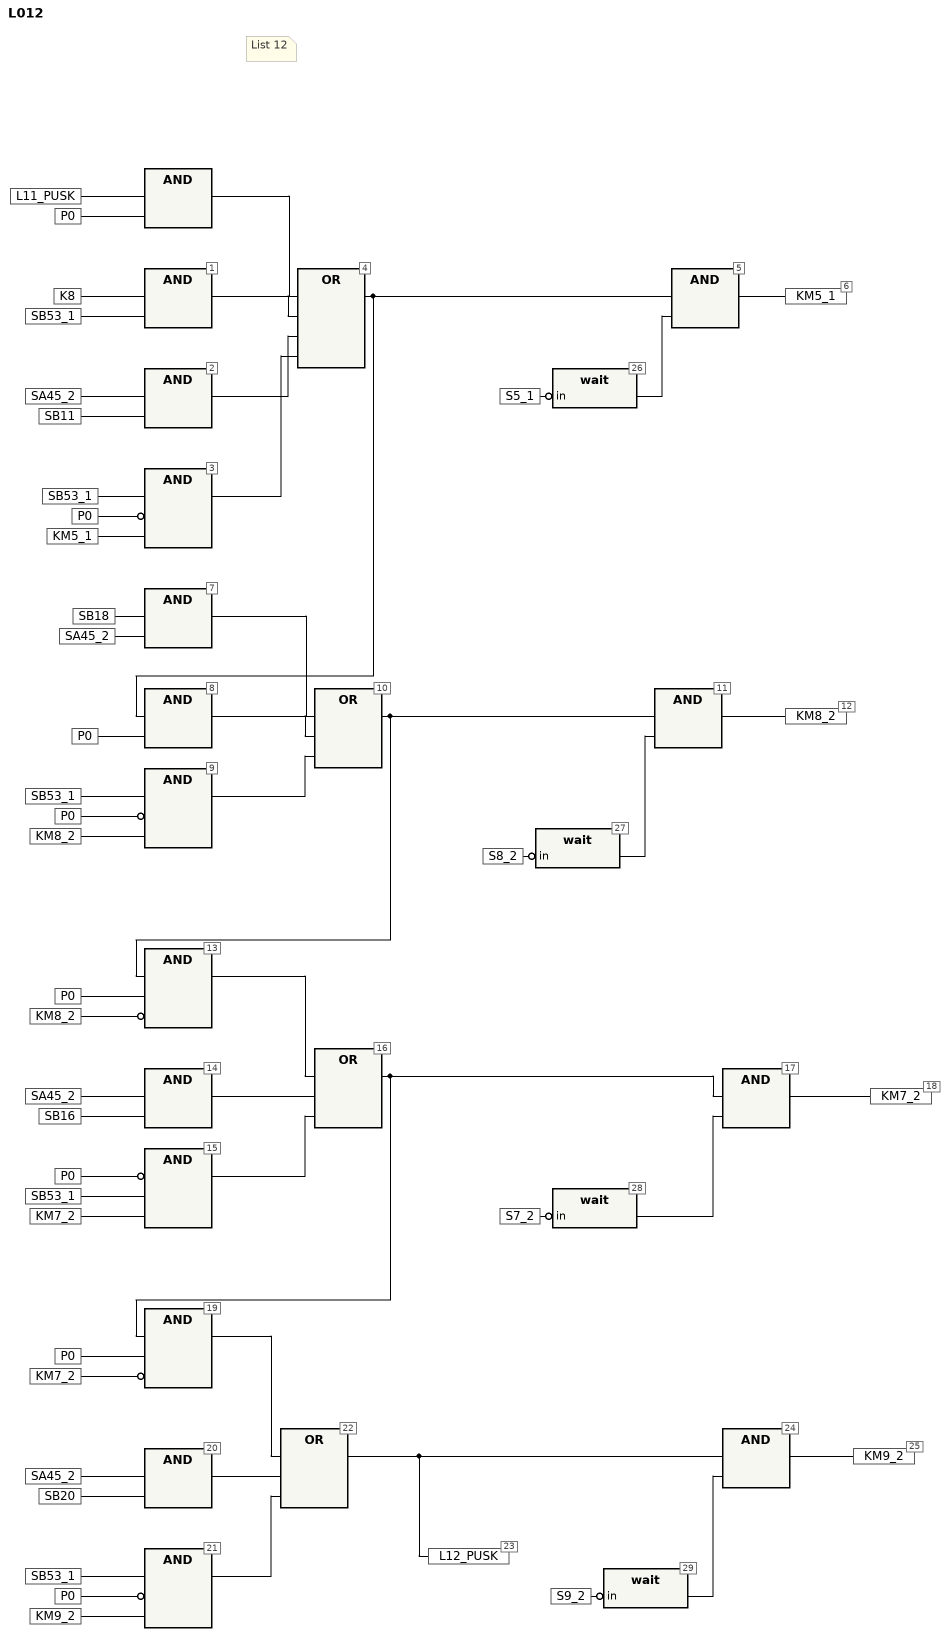
_CFC_ (* Continuous Function Chart, elements in execution order *)
(* List 12 *)
#0 AND(L11_PUSK, P0)
#1 AND(K8, SB53_1)
#2 AND(SA45_2, SB11)
#3 AND(SB53_1, NOT P0, KM5_1)
#4 OR(#0, #1, #2, #3)
#5 AND(#4, #26)
#6 KM5_1 <= #5
#7 AND(SB18, SA45_2)
#8 AND(#4, P0)
#9 AND(SB53_1, NOT P0, KM8_2)
#10 OR(#7, #8, #9)
#11 AND(#10, #27)
#12 KM8_2 <= #11
#13 AND(#10, P0, NOT KM8_2)
#14 AND(SA45_2, SB16)
#15 AND(NOT P0, SB53_1, KM7_2)
#16 OR(#13, #14, #15)
#17 AND(#16, #28)
#18 KM7_2 <= #17
#19 AND(#16, P0, NOT KM7_2)
#20 AND(SA45_2, SB20)
#21 AND(SB53_1, NOT P0, KM9_2)
#22 OR(#19, #20, #21)
#23 L12_PUSK <= #22
#24 AND(#22, #29)
#25 KM9_2 <= #24
#26 wait(in: NOT S5_1)
#27 wait(in: NOT S8_2)
#28 wait(in: NOT S7_2)
#29 wait(in: NOT S9_2)
_END_CFC_
(* the same logic as Structured Text *)
(* List 12 *)
_t5 := (L11_PUSK AND P0) OR (K8 AND SB53_1) OR (SA45_2 AND SB11) OR (SB53_1 AND NOT P0 AND KM5_1);
KM5_1 := _t5 AND _t85;
_t25 := (SB18 AND SA45_2) OR (_t5 AND P0) OR (SB53_1 AND NOT P0 AND KM8_2);
KM8_2 := _t25 AND _t86;
_t45 := (_t25 AND P0 AND NOT KM8_2) OR (SA45_2 AND SB16) OR (NOT P0 AND SB53_1 AND KM7_2);
KM7_2 := _t45 AND _t87;
_t59 := (_t45 AND P0 AND NOT KM7_2) OR (SA45_2 AND SB20) OR (SB53_1 AND NOT P0 AND KM9_2);
L12_PUSK := _t59;
KM9_2 := _t59 AND _t88;
_t85 := wait(in := NOT S5_1);
_t86 := wait(in := NOT S8_2);
_t87 := wait(in := NOT S7_2);
_t88 := wait(in := NOT S9_2);
END_PROGRAM

(* POU L013, CFC *)
PROGRAM L013
VAR



	P4: BOOL;

END_VAR
VAR (* helpers for the ST form of the networks *)
	_t12 : BOOL;
	_t20 : BOOL;
	_t19 : BOOL;
	_t23 : BOOL;
END_VAR
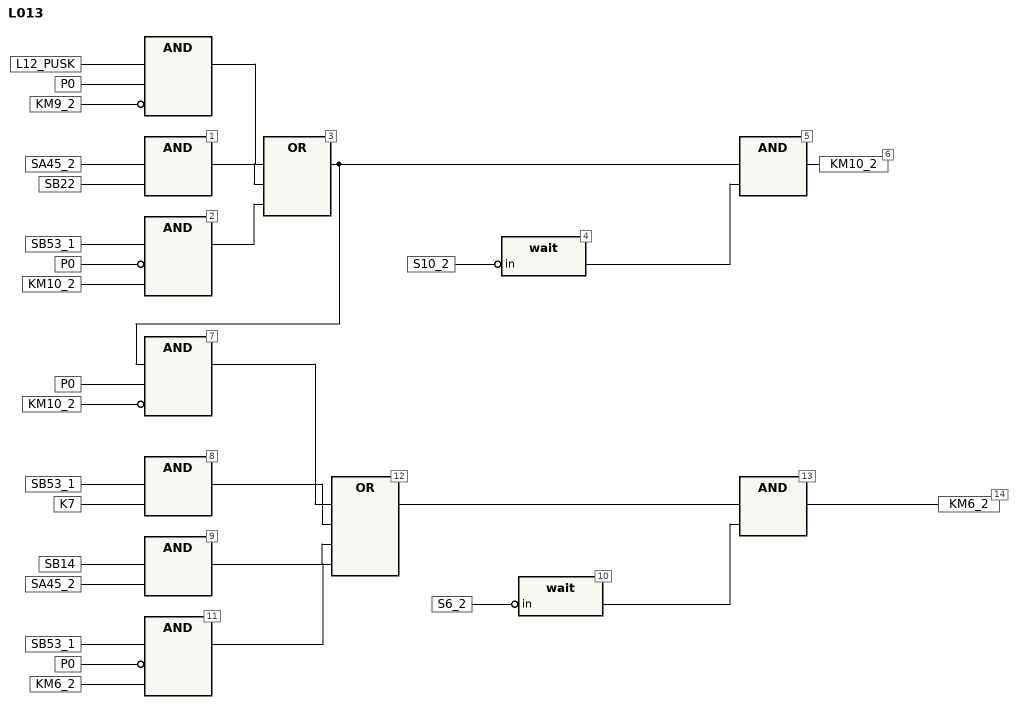
_CFC_ (* Continuous Function Chart, elements in execution order *)
#0 AND(L12_PUSK, P0, NOT KM9_2)
#1 AND(SA45_2, SB22)
#2 AND(SB53_1, NOT P0, KM10_2)
#3 OR(#0, #1, #2)
#4 wait(in: NOT S10_2)
#5 AND(#3, #4)
#6 KM10_2 <= #5
#7 AND(#3, P0, NOT KM10_2)
#8 AND(SB53_1, K7)
#9 AND(SB14, SA45_2)
#10 wait(in: NOT S6_2)
#11 AND(SB53_1, NOT P0, KM6_2)
#12 OR(#7, #8, #9, #11)
#13 AND(#12, #10)
#14 KM6_2 <= #13
_END_CFC_
(* the same logic as Structured Text *)
_t12 := (L12_PUSK AND P0 AND NOT KM9_2) OR (SA45_2 AND SB22) OR (SB53_1 AND NOT P0 AND KM10_2);
KM10_2 := _t12 AND wait(in := NOT S10_2);
_t20 := _t12 AND P0 AND NOT KM10_2;
_t19 := SB53_1 AND K7;
_t23 := SB14 AND SA45_2;
KM6_2 := (_t20 OR _t19 OR _t23 OR (SB53_1 AND NOT P0 AND KM6_2)) AND wait(in := NOT S6_2);
END_PROGRAM

(* POU L014, CFC *)
PROGRAM L014
VAR

END_VAR
VAR (* helpers for the ST form of the networks *)
	_t6 : BOOL;
	_t29 : BOOL;
END_VAR
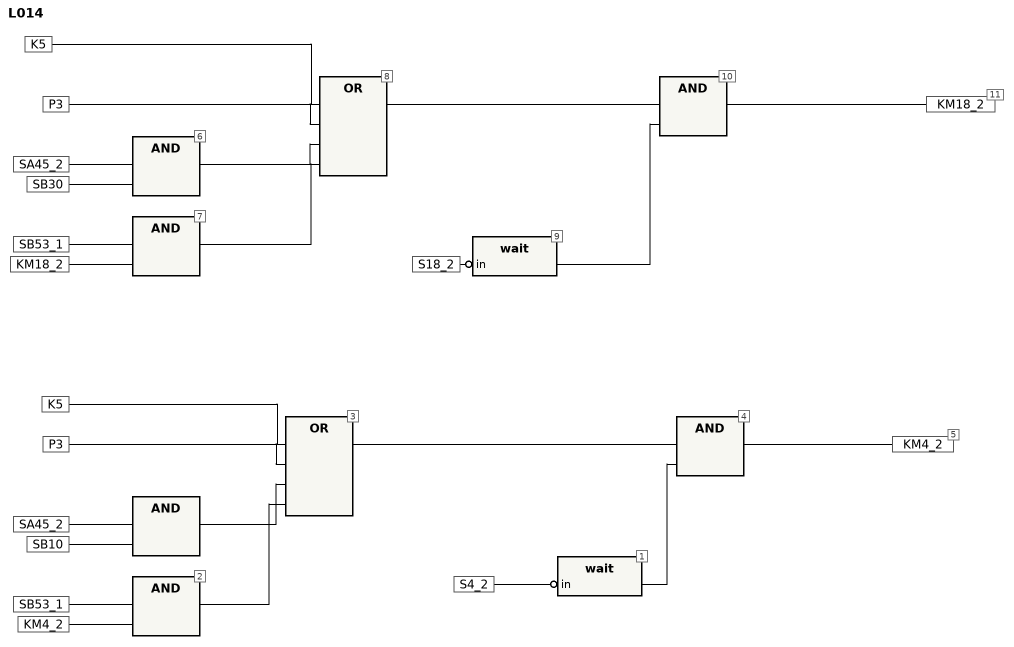
_CFC_ (* Continuous Function Chart, elements in execution order *)
#0 AND(SA45_2, SB10)
#1 wait(in: NOT S4_2)
#2 AND(SB53_1, KM4_2)
#3 OR(K5, P3, #0, #2)
#4 AND(#3, #1)
#5 KM4_2 <= #4
#6 AND(SA45_2, SB30)
#7 AND(SB53_1, KM18_2)
#8 OR(K5, P3, #6, #7)
#9 wait(in: NOT S18_2)
#10 AND(#8, #9)
#11 KM18_2 <= #10
_END_CFC_
(* the same logic as Structured Text *)
_t6 := SA45_2 AND SB10;
KM4_2 := (K5 OR P3 OR _t6 OR (SB53_1 AND KM4_2)) AND wait(in := NOT S4_2);
_t29 := K5 OR P3 OR (SA45_2 AND SB30) OR (SB53_1 AND KM18_2);
KM18_2 := _t29 AND wait(in := NOT S18_2);
END_PROGRAM

(* POU L015, CFC *)
PROGRAM L015
VAR

END_VAR
VAR (* helpers for the ST form of the networks *)
	_t14 : BOOL;
	_t20 : BOOL;
	_t28 : BOOL;
	_t34 : BOOL;
	_t46 : BOOL;
END_VAR
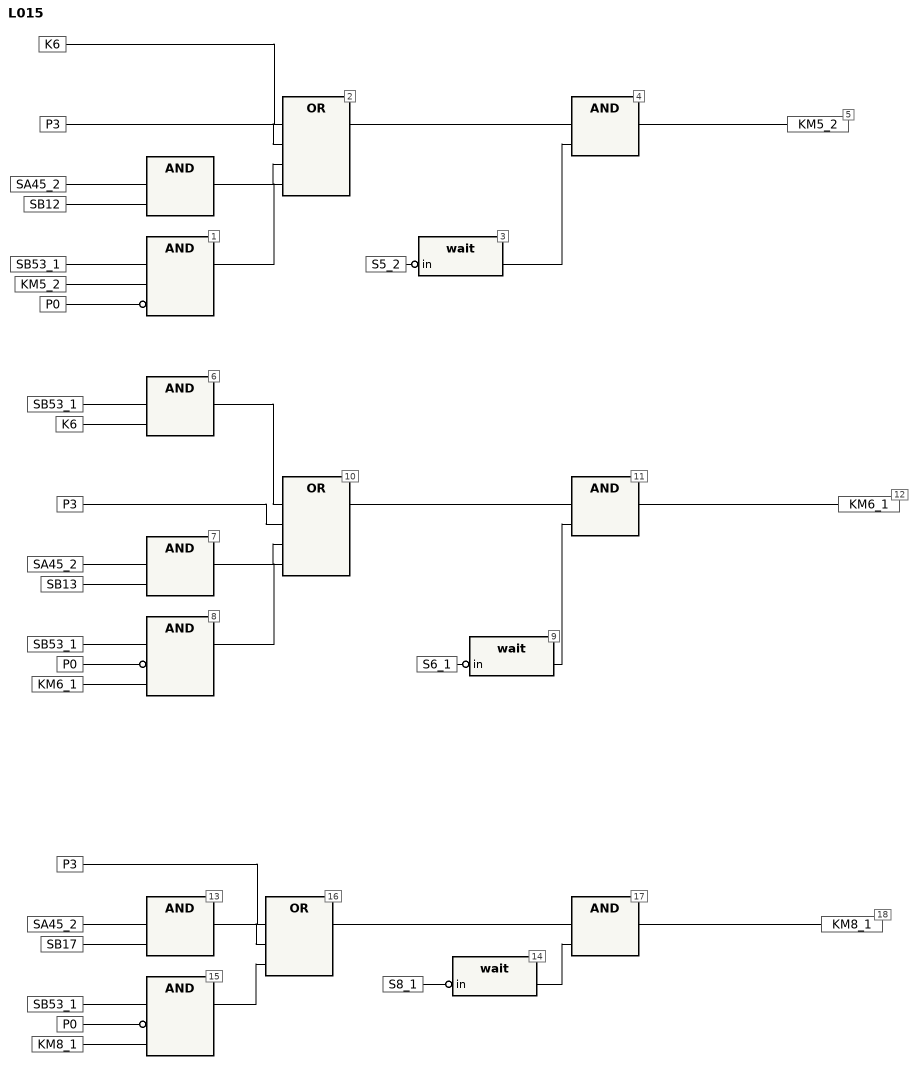
_CFC_ (* Continuous Function Chart, elements in execution order *)
#0 AND(SA45_2, SB12)
#1 AND(SB53_1, KM5_2, NOT P0)
#2 OR(K6, P3, #0, #1)
#3 wait(in: NOT S5_2)
#4 AND(#2, #3)
#5 KM5_2 <= #4
#6 AND(SB53_1, K6)
#7 AND(SA45_2, SB13)
#8 AND(SB53_1, NOT P0, KM6_1)
#9 wait(in: NOT S6_1)
#10 OR(#6, P3, #7, #8)
#11 AND(#10, #9)
#12 KM6_1 <= #11
#13 AND(SA45_2, SB17)
#14 wait(in: NOT S8_1)
#15 AND(SB53_1, NOT P0, KM8_1)
#16 OR(P3, #13, #15)
#17 AND(#16, #14)
#18 KM8_1 <= #17
_END_CFC_
(* the same logic as Structured Text *)
_t14 := K6 OR P3 OR (SA45_2 AND SB12) OR (SB53_1 AND KM5_2 AND NOT P0);
KM5_2 := _t14 AND wait(in := NOT S5_2);
_t20 := SB53_1 AND K6;
_t28 := SA45_2 AND SB13;
_t34 := SB53_1 AND NOT P0 AND KM6_1;
KM6_1 := (_t20 OR P3 OR _t28 OR _t34) AND wait(in := NOT S6_1);
_t46 := SA45_2 AND SB17;
KM8_1 := (P3 OR _t46 OR (SB53_1 AND NOT P0 AND KM8_1)) AND wait(in := NOT S8_1);
END_PROGRAM

(* POU L016, CFC *)
PROGRAM L016
VAR
	mt7TON: TON;

	mt9TON: TON;
	mt10TON: TON;
END_VAR
VAR (* helpers for the ST form of the networks *)
	_t3 : BOOL;
	_t51 : BOOL;
	_t81 : BOOL;
	_t96 : BOOL;
	_t126 : BOOL;
END_VAR
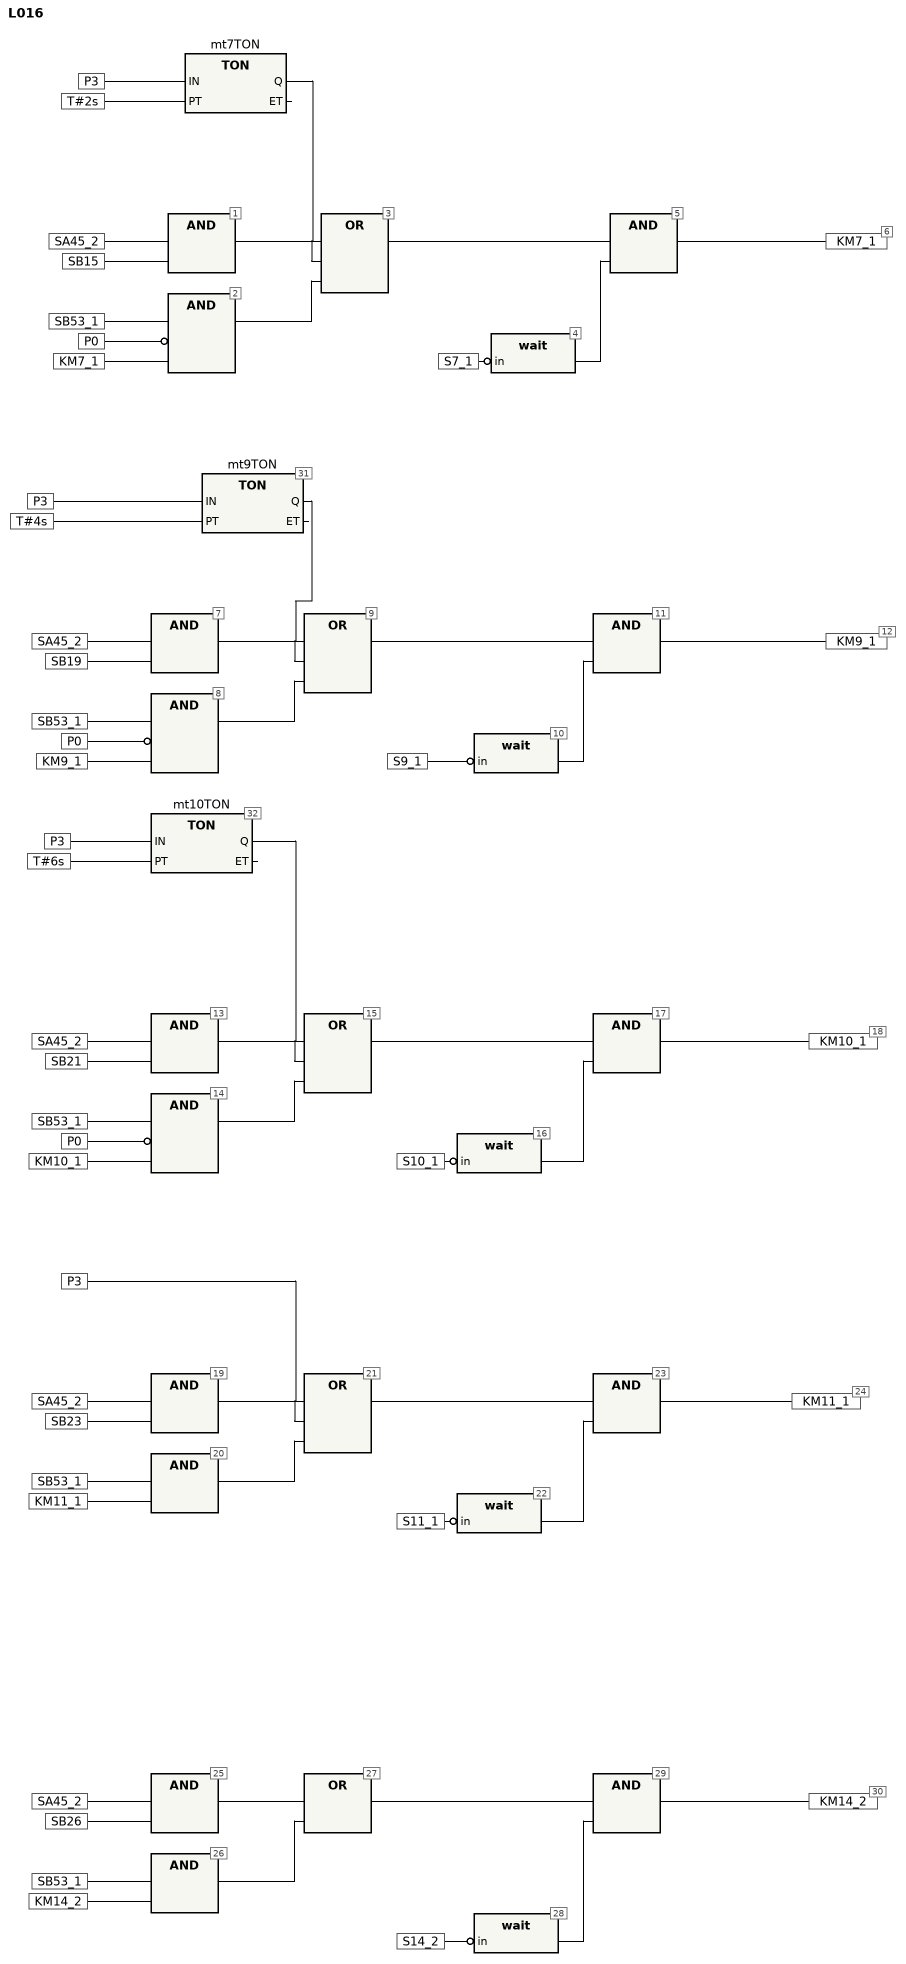
_CFC_ (* Continuous Function Chart, elements in execution order *)
#0 mt7TON:TON(IN: P3, PT: T#2s)
#1 AND(SA45_2, SB15)
#2 AND(SB53_1, NOT P0, KM7_1)
#3 OR(#0.Q, #1, #2)
#4 wait(in: NOT S7_1)
#5 AND(#3, #4)
#6 KM7_1 <= #5
#7 AND(SA45_2, SB19)
#8 AND(SB53_1, NOT P0, KM9_1)
#9 OR(#31.Q, #7, #8)
#10 wait(in: NOT S9_1)
#11 AND(#9, #10)
#12 KM9_1 <= #11
#13 AND(SA45_2, SB21)
#14 AND(SB53_1, NOT P0, KM10_1)
#15 OR(#32.Q, #13, #14)
#16 wait(in: NOT S10_1)
#17 AND(#15, #16)
#18 KM10_1 <= #17
#19 AND(SA45_2, SB23)
#20 AND(SB53_1, KM11_1)
#21 OR(P3, #19, #20)
#22 wait(in: NOT S11_1)
#23 AND(#21, #22)
#24 KM11_1 <= #23
#25 AND(SA45_2, SB26)
#26 AND(SB53_1, KM14_2)
#27 OR(#25, #26)
#28 wait(in: NOT S14_2)
#29 AND(#27, #28)
#30 KM14_2 <= #29
#31 mt9TON:TON(IN: P3, PT: T#4s)
#32 mt10TON:TON(IN: P3, PT: T#6s)
_END_CFC_
(* the same logic as Structured Text *)
mt7TON(IN := P3, PT := T#2s);
_t3 := mt7TON.Q OR (SA45_2 AND SB15) OR (SB53_1 AND NOT P0 AND KM7_1);
KM7_1 := _t3 AND wait(in := NOT S7_1);
_t51 := mt9TON.Q OR (SA45_2 AND SB19) OR (SB53_1 AND NOT P0 AND KM9_1);
KM9_1 := _t51 AND wait(in := NOT S9_1);
_t81 := mt10TON.Q OR (SA45_2 AND SB21) OR (SB53_1 AND NOT P0 AND KM10_1);
KM10_1 := _t81 AND wait(in := NOT S10_1);
_t96 := P3 OR (SA45_2 AND SB23) OR (SB53_1 AND KM11_1);
KM11_1 := _t96 AND wait(in := NOT S11_1);
_t126 := (SA45_2 AND SB26) OR (SB53_1 AND KM14_2);
KM14_2 := _t126 AND wait(in := NOT S14_2);
mt9TON(IN := P3, PT := T#4s);
mt10TON(IN := P3, PT := T#6s);
END_PROGRAM

(* Visualisation main
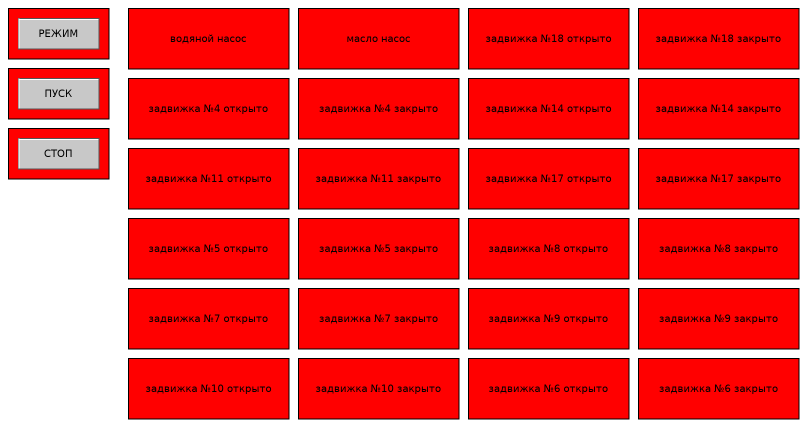
rounded rectangle at (130,10)-(291,71): text "водяной насос"; alarm colour if .KM1
rounded rectangle at (300,10)-(461,71): text "масло насос"; alarm colour if .KM2
rounded rectangle at (470,10)-(631,71): text "задвижка №18 открыто"; alarm colour if .KM18_1
rounded rectangle at (640,10)-(801,71): text "задвижка №18 закрыто"; alarm colour if .KM18_2
rounded rectangle at (130,80)-(291,141): text "задвижка №4 открыто"; alarm colour if .KM4_1
rounded rectangle at (300,80)-(461,141): text "задвижка №4 закрыто"; alarm colour if ._4gate.closed
rounded rectangle at (470,80)-(631,141): text "задвижка №14 открыто"; alarm colour if ._14gate.opened
rounded rectangle at (640,80)-(801,141): text "задвижка №14 закрыто"; alarm colour if ._14gate.closed
rounded rectangle at (130,150)-(291,211): text "задвижка №11 открыто"; alarm colour if ._11gate.opened
rounded rectangle at (300,150)-(461,211): text "задвижка №11 закрыто"; alarm colour if ._11gate.closed
rounded rectangle at (470,150)-(631,211): text "задвижка №17 открыто"; alarm colour if ._17gate.opened
rounded rectangle at (640,150)-(801,211): text "задвижка №17 закрыто"; alarm colour if ._17gate.closed
rounded rectangle at (130,220)-(291,281): text "задвижка №5 открыто"; alarm colour if ._5gate.opened
rounded rectangle at (300,220)-(461,281): text "задвижка №5 закрыто"; alarm colour if ._5gate.closed
rounded rectangle at (470,220)-(631,281): text "задвижка №8 открыто"; alarm colour if ._8gate.opened
rounded rectangle at (640,220)-(801,281): text "задвижка №8 закрыто"; alarm colour if ._8gate.closed
rounded rectangle at (130,290)-(291,351): text "задвижка №7 открыто"; alarm colour if ._7gate.opened
rounded rectangle at (300,290)-(461,351): text "задвижка №7 закрыто"; alarm colour if ._7gate.closed
rounded rectangle at (470,290)-(631,351): text "задвижка №9 открыто"; alarm colour if ._9gate.opened
rounded rectangle at (640,290)-(801,351): text "задвижка №9 закрыто"; alarm colour if ._9gate.closed
rounded rectangle at (130,360)-(291,421): text "задвижка №10 открыто"; alarm colour if ._10gate.opened
rounded rectangle at (300,360)-(461,421): text "задвижка №10 закрыто"; alarm colour if ._10gate.closed
rounded rectangle at (470,360)-(631,421): text "задвижка №6 открыто"; alarm colour if ._6gate.opened
rounded rectangle at (640,360)-(801,421): text "задвижка №6 закрыто"; alarm colour if ._6gate.closed
rounded rectangle at (10,130)-(111,181): alarm colour if .goSTOP
button at (20,140)-(101,171): text "СТОП"; toggles .SB53_1
rounded rectangle at (10,70)-(111,121): alarm colour if .goPusk
button at (20,80)-(101,111): text "ПУСК"; toggles .SB43
rounded rectangle at (10,10)-(111,61): alarm colour if .goRejim
button at (20,20)-(101,51): text "РЕЖИМ"; toggles .SB42
*)
